Universal Robots PolyScope program: remote_control_2.urp

Program remote_control_2 (createdIn=5.0.4.30603 lastSavedIn=5.0.4.30603 robotSerialNumber=20185500075 directory=/programs/usbdisk installation=default)
Calibrated DH parameters: a=[0.00014, -0.411556, -0.391866, 0.000087, 0.000022, 0]; d=[0.162531, 44.696176, -48.162844, 3.60009, 0.099865, 0.099717]; alpha=[1.57034, -0.002382, 0.004778, 1.570459, -1.570578, 0]; deltaTheta=[0, -0.253176, 6.494118, 0.042247, 0.000001, 0]
BeforeStart
  host := socket_open("129.78.210.145", 30000)
  initialising := 1
Robot Program (runOnlyOnce=true motionType=MoveJ speed=0 acceleration=0 useActiveTCP=true positionType=CartesianPose)
  Loop While (checkContinuously=false) expression=host≟False
    host := socket_open("129.78.210.145", 30000)
    Wait Sleep waitTime=0.1
  success := socket_send_string("Shaking hands")
  Wait Sleep waitTime=0.05
  new_waypts_flag := 0
  initialising := 0
  Script file /programs/usbdisk/client_move.script
    | waypoints=[0,0,0,0,0,0,0,0,0,0,0,0,0,0,0,0,0,0,0,0,0,0,0,0,0,0,0,0,0,0,0]
    | num_waypoints=0
    | 
    | while 1:
    | 
    | if new_waypts_flag==1:
    |  waypoints=new_waypts
    |  num_waypoints=waypoints[0]
    |  new_waypts_flag=0
    | end
    | 
    | i=1
    | while i<= num_waypoints:
    |   joints = [waypoints[i], waypoints[i+1], waypoints[i+2], waypoints[i+3], waypoints[i+4], waypoints[i+5]]
    |   movep(joints, v=0.05, r=0.1)
    |   i=i+6
    | end
    | 
    | if num_waypoints==0:
    |  sleep(0.01)
    | end
    | 
    | end
Thread Thread_1 (runOnlyOnce=false trackProgramExecution=false)
  Loop While (checkContinuously=false) expression=initialising≟1
    Wait Sleep waitTime=0.01
  Loop Forever
    new_waypts_flag := 0
    new_waypts := socket_read_ascii_float(30)
    If new_waypts[0]≠0
      new_waypts_flag := 1
      Wait Condition expression=new_waypts_flag≟0
      success := socket_send_string("ready")
    Wait Sleep waitTime=0.01
